(*********************************** G.D S.p.A. - Technical Department ***********************************
============= PROGRAM INFO ============
FOLDER:             TBD
MACHINES INVOLVED:  TBD 

============= DESCRIPTION =============
csp machine declaration

============= REVISIONS ===============
Date		Version	 	Author      	Description             
----------	-------		------------  	--------------------------------------------
2019/04/05 	0000.00	 	M.Grasso		Creation of the PRG

**********************************************************************************************************)
(*$R process_ref := prc; $*)
PROGRAM csp_case_feed_reject_belt
VAR
		
	prc:											process;
	prc_path:										STRING;
	
END_VAR

_read_var_input();

_object_manager();

IF NOT objects_running()
THEN
	RETURN;	
END_IF

_read_process_image();

_mode_manager();

_set_runtime_properties();

(********************************* BODY *********************************)
(************************************************************************)

_handle_messages();

_write_output();

ACTION _handle_messages:
;
END_ACTION

ACTION _handle_process_test:
;
END_ACTION

ACTION _mode_manager:
IF process_mode_req_is_pending(prc)
THEN
    process_apply_mode_req_first_step(prc);
    CASE process_get_mode(prc) OF
        MODE_TO_ABSENT:
			;
        MODE_TO_INACTIVE:
			;
        MODE_TO_TEST:
			;
        MODE_TO_OPERATIONAL:
			;
    END_CASE
    process_apply_mode_req_second_step(prc);
END_IF
END_ACTION

ACTION _object_manager:
IF objects_initialization()
THEN
	sub_process_init(
		object_name					:= 'csp_case_feed_reject_belt.prc', 
		process						:= csp_case_feed_reject.prc, 
		CONVERSION_this				:= prc);
		
	prc_path 						:= process_get_path(prc);
END_IF

IF objects_running()
THEN
	process_cycle(prc);
END_IF
END_ACTION

ACTION _read_process_image:
;
END_ACTION

ACTION _read_var_input:
;
END_ACTION

ACTION _set_runtime_properties:
;
END_ACTION

ACTION _write_output:
;
END_ACTION

END_PROGRAM

(* stored: Version 1.1.0.1, ProductVersion 3.1.4022.12
   POU csp_case_feed_reject_belt: Id {a6fdd87c-4931-452d-ac48-58b52833be44}, SpecialFunc None
   Action _handle_messages: Id {c973dab4-0d80-4fc5-a387-cfa126f240b6}
   Action _handle_process_test: Id {57a407a8-d13b-4882-b728-6a4d36416ca2}
   Action _mode_manager: Id {040c8676-7663-4676-99ac-a013e5ab0e48}
   Action _object_manager: Id {3b79fde1-df66-4589-9127-bb0da038fbc5}
   Action _read_process_image: Id {c72ef217-2168-4e33-b381-1afa6a05e8c2}
   Action _read_var_input: Id {7f2d7ed6-b8f5-4ae2-8a01-0eef23128ffa}
   Action _set_runtime_properties: Id {6d302c09-09ee-4fbd-a198-d371efd3df3a}
   Action _write_output: Id {21b506f2-89fa-49f0-b822-81af30ca597e} *)
